(* IEC 61131-3 sources: kebaiectestproject/system, 1 file *)

(* ---- systemAB.pu ---- *)
ALGORITHM_BLOCK systemAB #DUMMY_EDIT_BLOCK

SYSTEM_VAR
 sv_Bool : BOOL;
 sv_endless : BOOL;
END_VAR

SYSTEM_OBJECT
 TaskPU : TASK;
 TaskFast : TASK;
 TaskSlow : TASK;
END_OBJECT

VAR
 dummy : DINT;
 iCount : LINT;
 cnt : DINT;
 localBool : BOOL := FALSE;
END_VAR

POSTUPDATE_ALGORITHM Fehlersituation ON TaskPU WITH sv_Bool

#BEGIN_EDIT_BLOCK
dummy := Print("Post Update Triggered");

;#END_EDIT_BLOCK END_ALGORITHM

PROCESS_ALGORITHM setTrue ON TaskFast AUTOSTART

#BEGIN_EDIT_BLOCK
sv_Bool := TRUE;

;#END_EDIT_BLOCK END_ALGORITHM

PROCESS_ALGORITHM cyclicCompare ON TaskSlow AUTOSTART

#BEGIN_EDIT_BLOCK

IF sv_endless = TRUE THEN

FOR iCount := 1 TO 100000000 DO

   IF sv_Bool <> localBool THEN
      cnt := cnt + 1;
   END_IF;

END_FOR;

END_IF;

;#END_EDIT_BLOCK END_ALGORITHM

END_ALGORITHM_BLOCK

#END_OF_IEC_PART

@Puma @IecEditor 6 180 @Pou 25
@@@BEG_Comment@@@

@@@END_Comment@@@

@BEG_Contents

@BEG_Func
@RT(17)FuncTreeContainer
0
@END_Func

@BEG_Const
@RT(18)ConstTreeContainer
0
@END_Const

@BEG_Export

@BEG_Kind
@ALGORITHM_BLOCK @RT(8)systemAB @STRUCTURED_TEXT
@RT(0) @RT(0) @RT(0)
@END_Kind

@BEG_Dcl
@RT(16)DclTreeContainer
9
@Var @RT(7)sv_Bool @RT(0) @T @F @DT @RT(4)BOOL @RT(0) @T @T @BASIC 0 @F
@F @F
@T
@BEG_Attrib
3 @RT(0) @RT(0) @RT(0)
@END_Attrib
1 8 @F @F @F @F

@Var @RT(6)TaskPU @RT(0) @T @F @DT @RT(4)TASK @RT(0) @T @T @BASIC 0 @F
@F @F
@T
@BEG_Attrib
3 @RT(0) @RT(0) @RT(0)
@END_Attrib
1 7 @F @F @F @F

@Var @RT(8)TaskFast @RT(0) @T @F @DT @RT(4)TASK @RT(0) @T @T @BASIC 0 @F
@F @F
@T
@BEG_Attrib
3 @RT(0) @RT(0) @RT(0)
@END_Attrib
1 7 @F @F @F @F

@Var @RT(8)TaskSlow @RT(0) @T @F @DT @RT(4)TASK @RT(0) @T @T @BASIC 0 @F
@F @F
@T
@BEG_Attrib
3 @RT(0) @RT(0) @RT(0)
@END_Attrib
1 7 @F @F @F @F

@Var @RT(5)dummy @RT(0) @T @F @DT @RT(4)DINT @RT(0) @T @T @BASIC 0 @F
@F @F
@T
@BEG_Attrib
3 @RT(0) @RT(0) @RT(0)
@END_Attrib
1 0 @F @F @F @F

@Var @RT(6)iCount @RT(0) @T @F @DT @RT(4)LINT @RT(0) @T @T @BASIC 0 @F
@F @F
@T
@BEG_Attrib
3 @RT(0) @RT(0) @RT(0)
@END_Attrib
1 0 @F @F @F @F

@Var @RT(3)cnt @RT(0) @T @F @DT @RT(4)DINT @RT(0) @T @T @BASIC 0 @F
@F @F
@T
@BEG_Attrib
3 @RT(0) @RT(0) @RT(0)
@END_Attrib
1 0 @F @F @F @F

@Var @RT(9)localBool @RT(0) @T @F @DT @RT(4)BOOL @RT(0) @T @T @BASIC 0 @F
@F @F
@T
@BEG_Attrib
3 @RT(5)FALSE @RT(0) @RT(0)
@END_Attrib
1 0 @F @F @F @F

@Var @RT(10)sv_endless @RT(0) @T @F @DT @RT(4)BOOL @RT(0) @T @T @BASIC 0 @F
@F @F
@T
@BEG_Attrib
3 @RT(0) @RT(0) @RT(0)
@END_Attrib
1 8 @F @F @F @F

@END_Dcl

@END_Export

@BEG_Body

3

@BEG_Export

@BEG_Algo
@POSTUPDATE_ALGORITHM @RT(15)Fehlersituation @STRUCTURED_TEXT
@RT(0) @RT(7)sv_Bool @RT(6)TaskPU @F @F
@END_Algo

@BEG_Dcl
@RT(16)DclTreeContainer
0
@END_Dcl

@END_Export

@BEG_Export

@BEG_Algo
@PROCESS_ALGORITHM @RT(7)setTrue @STRUCTURED_TEXT
@RT(0) @RT(0) @RT(8)TaskFast @T @F
@END_Algo

@BEG_Dcl
@RT(16)DclTreeContainer
0
@END_Dcl

@END_Export

@BEG_Export

@BEG_Algo
@PROCESS_ALGORITHM @RT(13)cyclicCompare @STRUCTURED_TEXT
@RT(0) @RT(0) @RT(8)TaskSlow @T @F
@END_Algo

@BEG_Dcl
@RT(16)DclTreeContainer
0
@END_Dcl

@END_Export

@BEG_Body
@TL(2)
dummy := Print("Post Update Triggered");

@END_Body

@@@BEG_Comment@@@
@TL(0)

@@@END_Comment@@@

@BEG_Body
@TL(2)
sv_Bool := TRUE;

@END_Body

@@@BEG_Comment@@@
@TL(0)

@@@END_Comment@@@

@BEG_Body
@TL(15)

IF sv_endless = TRUE THEN

FOR iCount := 1 TO 100000000 DO

   IF sv_Bool <> localBool THEN
      cnt := cnt + 1;
   END_IF;

END_FOR;

END_IF;

@END_Body

@@@BEG_Comment@@@
@TL(0)

@@@END_Comment@@@
@END_Body

@END_Contents
